(*
Description: Models the transducers used for wicket gate differential 
			 pressure testing. FB methods take the input voltage from
			 EL3104 card and converts it to a PSIG pressure from 0-3000 PSIG.
			 Transducer pressure vs. voltage characteristic curve was tested and
			 found to be linear. See tranducer nameplate for detailed specs. 

METHODS: 	(1) PressureReading : REAL => Takes voltage reading and converts to pressure (PSIG.

Note: 		(1) Any method returning a value of -1 means an error occured

Author: Labib K. 
Engineering Co-op Student (2024)
August 9th, 2024
*)

FUNCTION_BLOCK PressureTransducer_3000PSIG

VAR CONSTANT
	nMaxRatedPressure : UINT := 3000;// PSIG
	nMaxVoltage : UINT := 10; // Volts
	nDefaultDAQ_startVal : INT := 6540;
	rDefaultEU_startVal : REAL := 0.0; //Volts
END_VAR

VAR_INPUT
	nDAQ_inputVoltage : REAL; //Links GVL.rVoltage_InputX
	rStartValInput_EU : REAL;
	nStartValInput : INT; 
END_VAR

VAR
	rStartVal_EU : REAL; //Engineering start value
	nStartVal : INT; //El3104 DAQ resolution, 16 bit (1 bit = sign bit)
	rTransducerVoltage : REAL; //Made local scope of object for accessibility later
END_VAR

//check whether SC works

(*
Descriptions of what each line does in the execution plane

1 => IF NOT zero, rStartVal_EU = User defined, ELSE takes default value OF 0 V
2 => If not zero, rStartVal = User defined, else takes default value of 6540
*)
VAR // added by the converter: edge detectors and wires of the graphical bodies
    _w1, _w2 : BOOL;
END_VAR

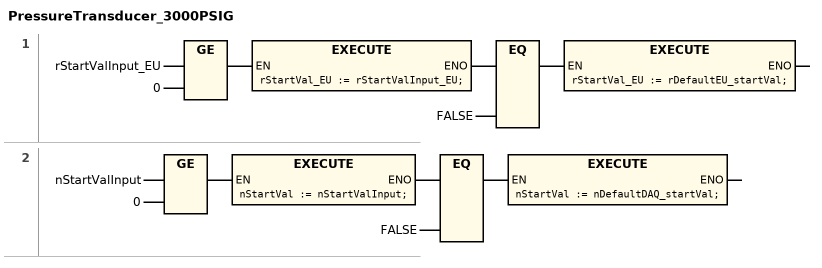
// NETWORK 1
_w1 := rStartValInput_EU >= 0;
IF _w1 THEN rStartVal_EU := rStartValInput_EU; END_IF
IF _w1 = FALSE THEN rStartVal_EU := rDefaultEU_startVal; END_IF

// NETWORK 2
_w2 := nStartValInput >= 0;
IF _w2 THEN nStartVal := nStartValInput; END_IF
IF _w2 = FALSE THEN nStartVal := nDefaultDAQ_startVal; END_IF

(*
Purpose: Converts the voltage signal from the pressure transducer into a pressure.
		 Firstly by converting the DAQ input signed 16 bit number to voltage, then convert voltage to PSIG
		 using linear interpolation

NOTE: The El3104 can only tolerate +/- 10V and a max input current of 40mA.

Inputs:     (1) rStartValInput_EU : REAL => User defined startValue_EU, set to zero to use default value of 0V (TEST PLZ LK)
		    (2) nStartValInput : INT => User defined startValue, set to zero to use default value of 6540 (unitless)

GVL usage:  (1) nVoltage_Input1 : INT => RAW current signed 16 bit voltage data from DAQ in terminal slot I1
		    (2) rVoltage_Input1_EU : REAL => Converted DAQ reading to voltage

Author: Labib K. 
Engineering Co-op Student (2024)
August 9th, 2024
*)

METHOD PUBLIC PressureReading : REAL
VAR
	rDAQtoVoltage : REAL; //DAQ signed 16 bit number to EU (V)
	rVoltToPSIG : REAL; //Conversion factor from volts to PSIG
END_VAR

//Comment to check whether SC is working

(*
Descriptions of what each line does in the execution plane

1 => Calculates Conversion factor DAQ resolution to V
2 => Multiplies raw DAQ resolution (unit less) -> Engineering unit(V) using linear interpolation
3 => Scales the Engineering Unit to a %Postion (4 mA = 0%)
4 => Reports the non-negative % Position, zero otherwise
*)
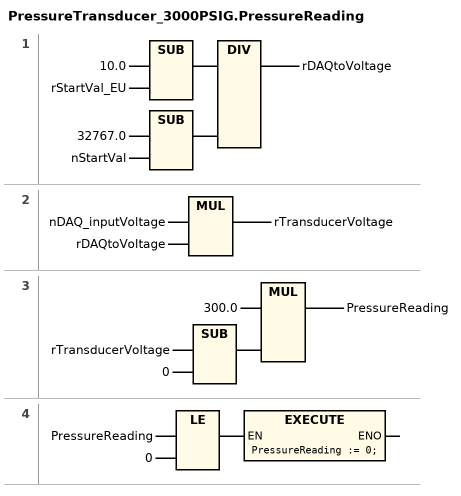
// NETWORK 1
rDAQtoVoltage := (10.0 - rStartVal_EU) / (32767.0 - nStartVal);

// NETWORK 2
rTransducerVoltage := nDAQ_inputVoltage * rDAQtoVoltage;

// NETWORK 3
PressureReading := 300.0 * (rTransducerVoltage - 0);

// NETWORK 4
IF PressureReading <= 0 THEN PressureReading := 0; END_IF
END_METHOD

END_FUNCTION_BLOCK

(* stored: Version 1.1.0.1, ProductVersion 3.1.4024.12
   POU PressureTransducer_3000PSIG: Id {b9c4d1ea-3f22-402c-9280-87bcd4ccb2a8}, SpecialFunc None
   Method PressureReading: Id {17e1ad5b-7935-41ee-b7aa-83c0ec7b9118} *)
